// Mitsubishi GX Works2 project: ladder2   PLC: FX3U/FX3UC

PROGRAM MAIN
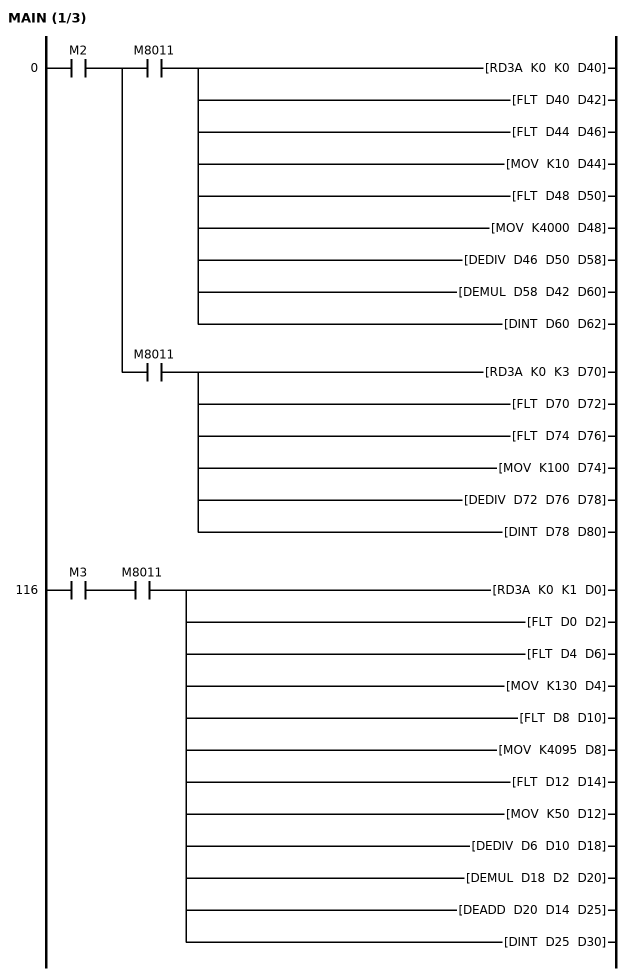
0     LD      M2
      MPS
      AND     M8011
      RD3A    K0 K0 D40
        [note] voltmeter
      FLT     D40 D42
      FLT     D44 D46
      MOV     K10 D44
      FLT     D48 D50
      MOV     K4000 D48
      DEDIV   D46 D50 D58
      DEMUL   D58 D42 D60
      DINT    D60 D62
      MPP
      AND     M8011
      RD3A    K0 K3 D70
        [note] ammeter
      FLT     D70 D72
      FLT     D74 D76
      MOV     K100 D74
      DEDIV   D72 D76 D78
      DINT    D78 D80
116   LD      M3
      AND     M8011
      RD3A    K0 K1 D0
        [note] NTC temp sensor
      FLT     D0 D2
      FLT     D4 D6
      MOV     K130 D4
      FLT     D8 D10
      MOV     K4095 D8
      FLT     D12 D14
      MOV     K50 D12
      DEDIV   D6 D10 D18
      DEMUL   D18 D2 D20
      DEADD   D20 D14 D25
      DINT    D25 D30
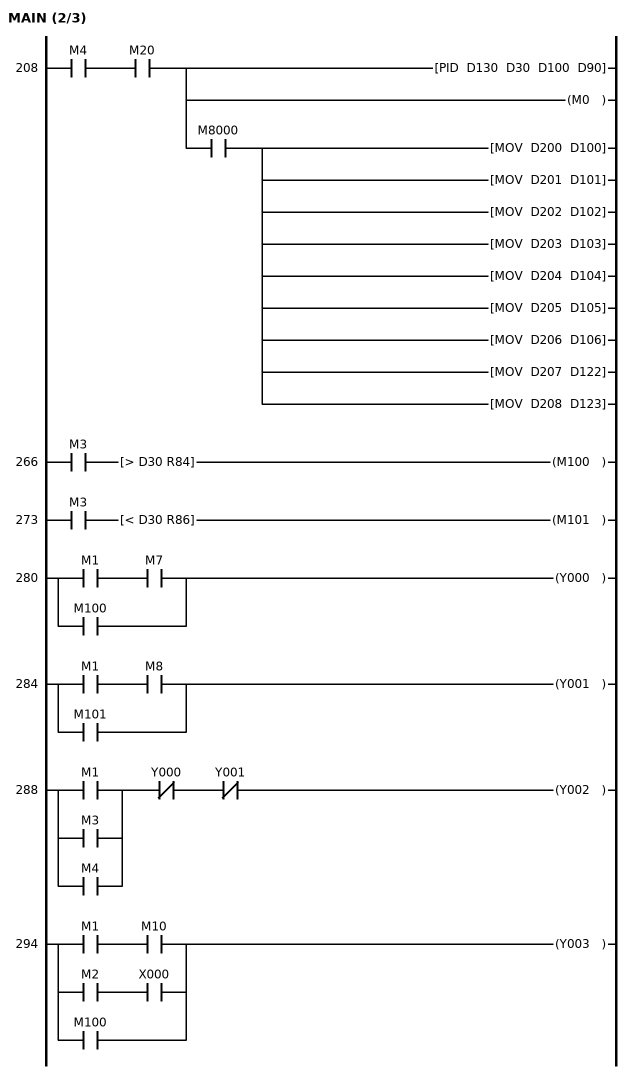
208   LD      M4
      AND     M20
      PID     D130 D30 D100 D90
        [note] PID Cotrol
      OUT     M0
      AND     M8000
      MOV     D200 D100
      MOV     D201 D101
      MOV     D202 D102
      MOV     D203 D103
      MOV     D204 D104
      MOV     D205 D105
      MOV     D206 D106
      MOV     D207 D122
      MOV     D208 D123
266   LD      M3
      AND>    D30 R84
      OUT     M100
        [note] high temp
273   LD      M3
      AND<    D30 R86
      OUT     M101
        [note] low temp
280   LD      M1
      AND     M7
      OR      M100
      OUT     Y000
        [note] red led
284   LD      M1
      AND     M8
      OR      M101
      OUT     Y001
        [note] blue led
288   LD      M1
      OR      M3
      OR      M4
      ANI     Y000
      ANI     Y001
      OUT     Y002
        [note] green led
294   LD      M1
      AND     M10
      LD      M2
      AND     X000
      ORB
      OR      M100
      OUT     Y003
        [note] cooler
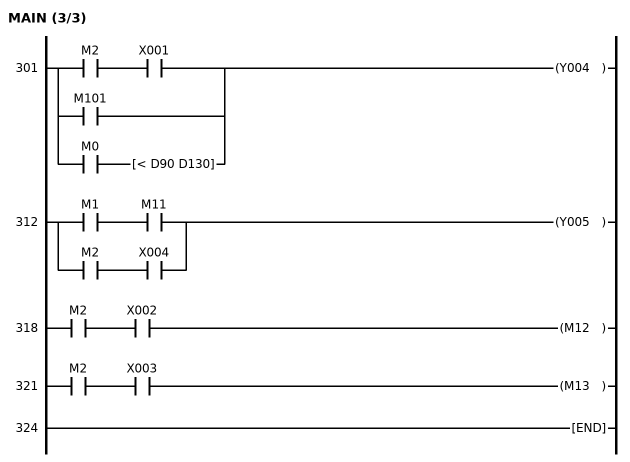
301   LD      M2
      AND     X001
      OR      M101
      LD      M0
      AND<    D90 D130
      ORB
      OUT     Y004
        [note] heater
312   LD      M1
      AND     M11
      LD      M2
      AND     X004
      ORB
      OUT     Y005
        [note] pump
318   LD      M2
      AND     X002
      OUT     M12
        [note] valve
321   LD      M2
      AND     X003
      OUT     M13
324   END
END_PROGRAM
